(* PLC project SafeLOGIC-1, BrAutomation SafeDESIGNER  4.4.1.0 *)
(* stored: companyURL http://www.br-automation.com, creationDateTime Sat Aug 05 11:09:40 2023 *)

PROGRAM Main

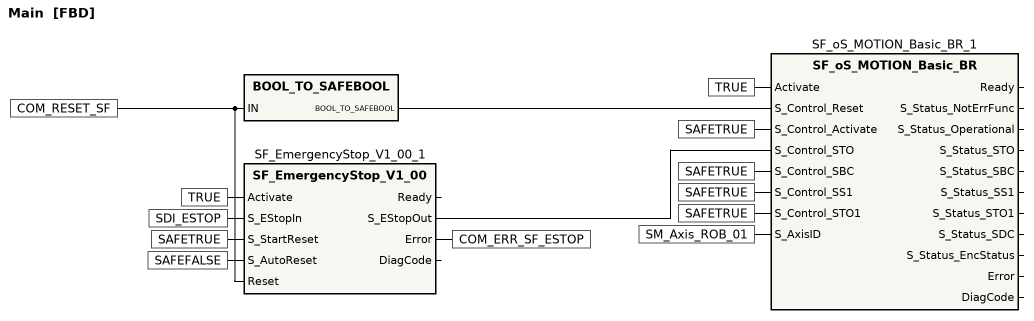
(* FBD diagram, written out as Structured Text *)
SF_EmergencyStop_V1_00_1(Activate := TRUE, S_EStopIn := SDI_ESTOP, S_StartReset := SAFETRUE, S_AutoReset := SAFEFALSE, Reset := COM_RESET_SF);
COM_ERR_SF_ESTOP := SF_EmergencyStop_V1_00_1.Error;
SF_oS_MOTION_Basic_BR_1(Activate := TRUE, S_Control_Reset := BOOL_TO_SAFEBOOL(COM_RESET_SF), S_Control_Activate := SAFETRUE, S_Control_STO := SF_EmergencyStop_V1_00_1.S_EStopOut, S_Control_SBC := SAFETRUE, S_Control_SS1 := SAFETRUE, S_Control_STO1 := SAFETRUE, S_AxisID := SM_Axis_ROB_01);
END_PROGRAM
